RoboDK station: Присоска.rdk

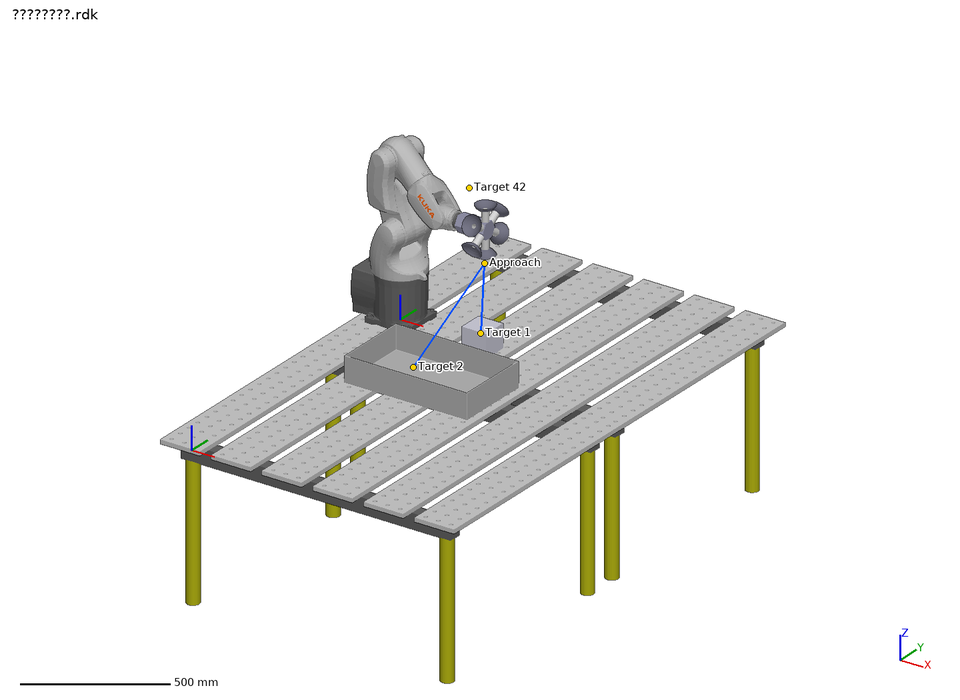
[picture v0: the station drawn from its stored meshes, robots at their saved joint values, targets as dots, program paths as lines]
Station ). Poses are relative to the parent item; angles as X-Y-Z fixed-axis rotations.
  - frame ABB IRB 120-3/0.6 Base at (60.92, -16.78, 0) mm
    - robot KUKA KR 3 R540: 6 axes, payload 3 kg, reach 541 mm, repeatability 0.02 mm, weight 26 kg
        modified DH rows (alpha deg, a mm, theta deg, d mm): 0, 0, 0, 345; -90, 20, 0, 0; 0, 260, -90, 0; -90, 20, 0, 260; 90, 0, 0, 0; -90, 0, 180, 75
        joint limits [-170, -170, -110, -175, -120, -350] to [170, 50, 155, 175, 120, 350]; home [0, -90, 90, 0, 0, 0]; saved at [9.598, -98.142, 138.557, 14.619, -41.348, -11.079]
      - tool TCP 1, TCP at (73.87, -0.56, 98.27) mm
      - tool Tool, TCP at (125, -3.56, 100) mm, rotated rx 0 ry 90 rz 0 deg, size 184.7 x 197.7 x 137.7 mm
    - target Target 2 (Cartesian target) at (314.02, -373.37, 60.32) mm, rotated rx -180 ry 0 rz -180 deg; joints [69.398, -15.49, 81.366, 71.063, -81.731, -22.743] of KUKA KR 3 R540
    - target Target 1 (Cartesian target) at (350.78, -35.53, 62.02) mm, rotated rx 180 ry 0 rz 180 deg; joints [10.307, -19.838, 133.471, 11.228, -113.229, 4.477] of KUKA KR 3 R540
    - frame Frame pick and place at (0, 0, 0) mm
      - object Table at (462.97, 233.54, 0) mm, size 1193.8 x 965.2 x 609.6 mm, geometry from welding_table.sld
    - target Approach (Cartesian target) at (366.38, -35.93, 324.04) mm, rotated rx 180 ry 0 rz 180 deg; joints [9.598, -98.142, 138.557, 14.619, -41.348, -11.079] of KUKA KR 3 R540
    - frame Frame 2 at (0, 0, 0) mm
      - object Table at (462.83, -721.33, 0) mm, size 1193.8 x 965.2 x 609.6 mm, geometry from welding_table.sld
      - object Box v1 at (120, -500, 0) mm, rotated rx 0 ry 0 rz 90 deg, size 300 x 500 x 100 mm, geometry from Box v1.stl
    - target Target 42 (Cartesian target) at (309.94, -45.15, 590.28) mm, rotated rx 180 ry 0 rz -180 deg; joints [17.127, -113.521, 87.539, -35.124, 30.788, 31.144] of KUKA KR 3 R540
    - frame KUKA KR 3 R540 Base at (0, -1210.12, 0) mm
  - program pick and place (14 instructions, listed below)
  - program Replace objects (1 instructions, listed below)
  - object box at (415.51, -49.57, 42.59) mm, size 100 x 100 x 100 mm, geometry from box.sld
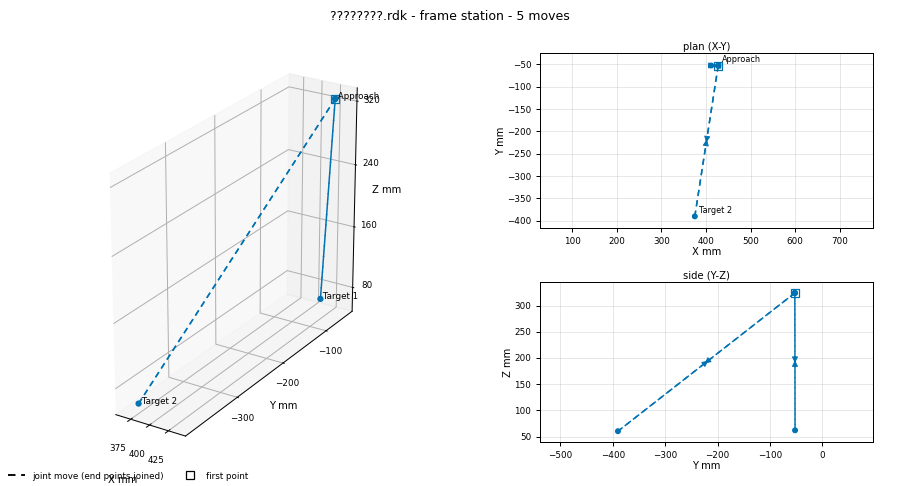
[picture p0: tool path of Присоска.rdk in frame station, 5 of 5 moves have a stored position in this frame; points joined in program order, loops and branches not executed]

--- program pick and place (robot KUKA KR 3 R540) ---
  Set speed (50.0 mm/s)
  Set Ref.: Frame pick and place
  Set Tool: Tool
  MoveJ (Approach)
  MoveJ (Target 1)
  Attach to Tool
  Call AirValve_On
  MoveJ (Approach)
  Change Frame -> Frame 2
  MoveJ (Target 2)
  Detach from Tool
  Call AirValve_Off
  MoveJ (Approach)
  Call Replace objects

--- program Replace objects (robot KUKA KR 3 R540) ---
  Replace objects
